TYPE UDT_HMI_FaultLogItem :
STRUCT
	sID : STRING;
	sDescription : STRING;
	sStartTime : STRING[19];
	sEndTime : STRING[19];
	dColor_Bg : DWORD := E_Color.White; // Table row background color
END_STRUCT
END_TYPE

(* stored: Version 1.1.0.1, ProductVersion 3.1.4024.11
   DUT UDT_HMI_FaultLogItem: Id {4fc01245-d77f-4454-90a8-2f14bfeac423} *)
